// TIA Portal project "Project_Axe" (V15)

(* hardware
DEVICE "HMI_1"  KTP400 Basic mono PN
   slot 0: "HMI_1"  KTP400 Basic mono PN  6AV6 647-0AA11-3AX0  12.0.0.0
   slot 1: "HMI_RT_1"  KTP400 Basic mono PN  6AV6 647-0AA11-3AX0  12.0.0.0
   slot 5: "HMI_1.IE_CP_1"  PROFINET Interface  12.0.0.0
      slot 1: "PROFINET Interface_1"  PROFINET Interface
         slot 1: "Port_1"  Port
DEVICE "S7-1200 station_1"  S7-1200 Station
   slot 0: "Rack_0"  S7-1200 Rack  Rack  V1.0
   slot 1: "PLC"  CPU 1212C AC/DC/Rly  6ES7 212-1BE31-0XB0  V3.0
*)

// ===== PLC "PLC"  CPU 1212C AC/DC/Rly =====

VAR_GLOBAL   // PLC tag table "Default tag table"
   "All_SelectionsCorrect" AT %I100.0 : Bool;
   "Stop" AT %I100.1 : Bool;
   "AxeBack" AT %Q100.0 : Bool;
   "TreeFall" AT %Q100.1 : Bool;
   "Reset" AT %Q100.2 : Bool;
   "SelectionsCorrectLight" AT %Q100.3 : Bool;
END_VAR

DATA_BLOCK "G"   // DB1
{ S7_Optimized_Access := 'TRUE' }
VERSION : 0.1
   VAR
      T1_DwellTime : IEC_TIMER;
      T2_AxeBack : IEC_TIMER;
      T3_AxeBounce : IEC_TIMER;
      T4_AxeSwing : IEC_TIMER;
      T5_TreeFall : IEC_TIMER;
      T6_WatchDog : IEC_TIMER;
      ResetTimeDelay : IEC_TIMER;
   END_VAR
   VAR RETAIN
      HMI_T1_Time : Real := 10.0;
      HMI_T2_Time : Real := 10.0;
      HMI_T3_Time : Real := 10.0;
      HMI_T4_Time : Real := 10.0;
      HMI_T5_Time : Real := 10.0;
      HMI_T6_Time : Real := 10.0;
   END_VAR
   VAR
      T1_Time : DInt;
      T2_Time : DInt;
      T3_Time : DInt;
      T4_Time : DInt;
      T5_Time : DInt;
      T6_Time : DInt;
   END_VAR
BEGIN
END_DATA_BLOCK

FUNCTION "Timers" : Void   // FC1, LAD
{ S7_Optimized_Access := 'TRUE' }
VERSION : 0.1
   VAR_TEMP
      temp_real1 : Real;
      temp_real2 : Real;
      temp_real4 : Real;
      temp_real3 : Real;
      temp_real5 : Real;
      temp_real6 : Real;
      temp_real_sum : Real;
   END_VAR
   VAR_TEMP   // added for the SCL form of the ladder/FBD networks
      _w1 : Bool;
   END_VAR
BEGIN

REGION Network 1: Dwell Time Before Starting Cycle
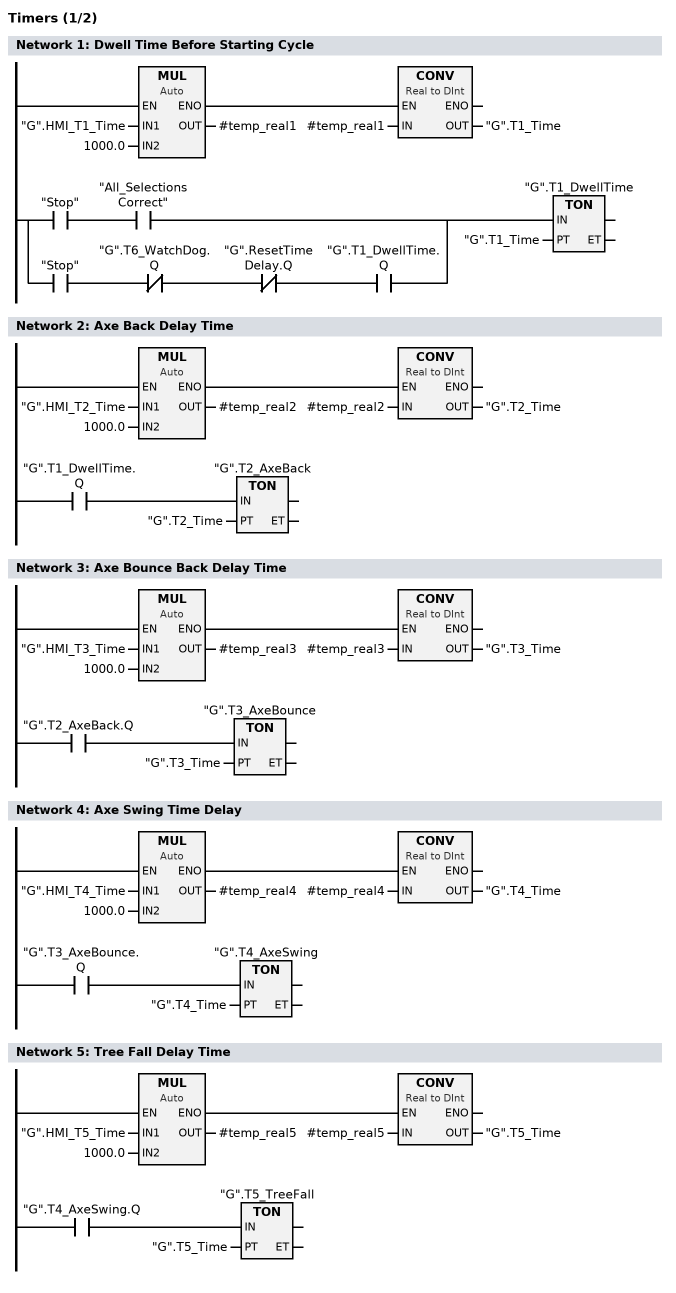
   // ENO of a box is taken as its EN; it also drops when the box reports an error
   #temp_real1 := "G".HMI_T1_Time * 1000.0;
   "G".T1_Time := REAL_TO_DINT(#temp_real1);
   "G".T1_DwellTime.TON(IN := ("Stop" AND "All_SelectionsCorrect") OR ("Stop" AND NOT "G".T6_WatchDog.Q AND NOT "G".ResetTimeDelay.Q AND "G".T1_DwellTime.Q),
                        PT := "G".T1_Time);
END_REGION

REGION Network 2: Axe Back Delay Time
   // ENO of a box is taken as its EN; it also drops when the box reports an error
   #temp_real2 := "G".HMI_T2_Time * 1000.0;
   "G".T2_Time := REAL_TO_DINT(#temp_real2);
   "G".T2_AxeBack.TON(IN := "G".T1_DwellTime.Q, PT := "G".T2_Time);
END_REGION

REGION Network 3: Axe Bounce Back Delay Time
   // ENO of a box is taken as its EN; it also drops when the box reports an error
   #temp_real3 := "G".HMI_T3_Time * 1000.0;
   "G".T3_Time := REAL_TO_DINT(#temp_real3);
   "G".T3_AxeBounce.TON(IN := "G".T2_AxeBack.Q, PT := "G".T3_Time);
END_REGION

REGION Network 4: Axe Swing Time Delay
   // ENO of a box is taken as its EN; it also drops when the box reports an error
   #temp_real4 := "G".HMI_T4_Time * 1000.0;
   "G".T4_Time := REAL_TO_DINT(#temp_real4);
   "G".T4_AxeSwing.TON(IN := "G".T3_AxeBounce.Q, PT := "G".T4_Time);
END_REGION

REGION Network 5: Tree Fall Delay Time
   // ENO of a box is taken as its EN; it also drops when the box reports an error
   #temp_real5 := "G".HMI_T5_Time * 1000.0;
   "G".T5_Time := REAL_TO_DINT(#temp_real5);
   "G".T5_TreeFall.TON(IN := "G".T4_AxeSwing.Q, PT := "G".T5_Time);
END_REGION

REGION Network 6: Watch Dog Delay Time. Summation of all times and the relay reset delay of 5 seconds
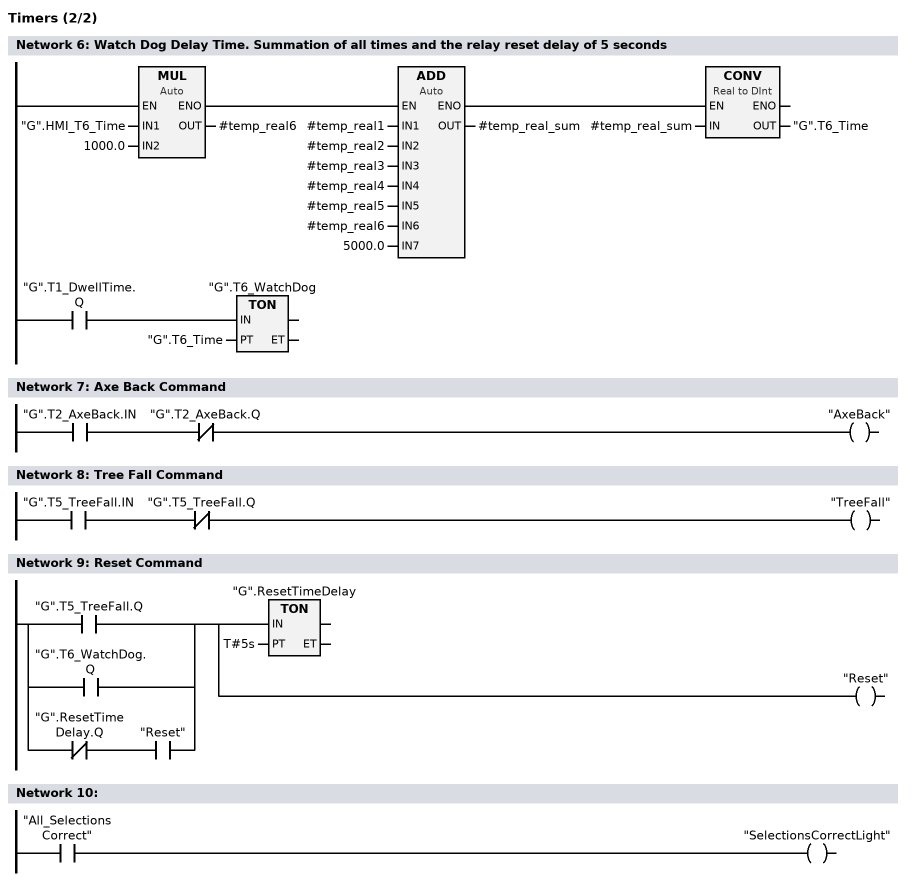
   // ENO of a box is taken as its EN; it also drops when the box reports an error
   #temp_real6 := "G".HMI_T6_Time * 1000.0;
   #temp_real_sum := #temp_real1 + #temp_real2 + #temp_real3 + #temp_real4 + #temp_real5 + #temp_real6 + 5000.0;
   "G".T6_Time := REAL_TO_DINT(#temp_real_sum);
   "G".T6_WatchDog.TON(IN := "G".T1_DwellTime.Q, PT := "G".T6_Time);
END_REGION

REGION Network 7: Axe Back Command
   RUNG wire#powerrail
      Contact( "G".T2_AxeBack.IN )
      I_Contact( "G".T2_AxeBack.Q )
      Coil( "AxeBack" )
   END_RUNG
   // the same network as SCL:
   "AxeBack" := "G".T2_AxeBack.IN AND NOT "G".T2_AxeBack.Q;
END_REGION

REGION Network 8: Tree Fall Command
   RUNG wire#powerrail
      Contact( "G".T5_TreeFall.IN )
      I_Contact( "G".T5_TreeFall.Q )
      Coil( "TreeFall" )
   END_RUNG
   // the same network as SCL:
   "TreeFall" := "G".T5_TreeFall.IN AND NOT "G".T5_TreeFall.Q;
END_REGION

REGION Network 9: Reset Command
   #_w1 := "G".T5_TreeFall.Q OR "G".T6_WatchDog.Q OR (NOT "G".ResetTimeDelay.Q AND "Reset");
   "G".ResetTimeDelay.TON(IN := #_w1, PT := T#5s);
   "Reset" := #_w1;
END_REGION

REGION Network 10
   RUNG wire#powerrail
      Contact( "All_SelectionsCorrect" )
      Coil( "SelectionsCorrectLight" )
   END_RUNG
   // the same network as SCL:
   "SelectionsCorrectLight" := "All_SelectionsCorrect";
END_REGION
END_FUNCTION

ORGANIZATION_BLOCK "Main"   // OB1, LAD, ProgramCycle
TITLE = "Main Program Sweep (Cycle)"
{ S7_Optimized_Access := 'TRUE' }
VERSION : 0.1
BEGIN

REGION Network 1
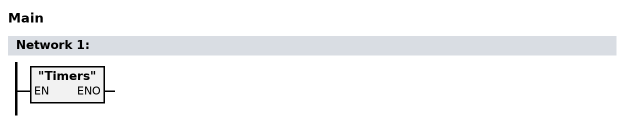
   RUNG wire#powerrail
      "Timers"()
   END_RUNG
   // the same network as SCL:
   "Timers"();
END_REGION
END_ORGANIZATION_BLOCK

(* ===== HMI "HMI_RT_1" =====
system functions are stored by id; their names below are inferred from use
connection "HMI_Connection_1": ETHERNET, SMART_S7_1200_OMS

HMI tags "Default tag table"
   "Tag_ScreenNumber" : UInt, internal
   "G_HMI_T1_Time" : Real = PLC G.HMI_T1_Time, 1 s
   "G_HMI_T2_Time" : Real = PLC G.HMI_T2_Time, 1 s
   "G_HMI_T3_Time" : Real = PLC G.HMI_T3_Time, 1 s
   "G_HMI_T4_Time" : Real = PLC G.HMI_T4_Time, 1 s
   "G_HMI_T5_Time" : Real = PLC G.HMI_T5_Time, 1 s
   "G_HMI_T6_Time" : Real = PLC G.HMI_T6_Time, 1 s
   "All_SelectionsCorrect" : Bool = PLC All_SelectionsCorrect AT %I100.0, 1 s
   "Stop" : Bool = PLC Stop AT %I100.1, 1 s
   "AxeBack" : Bool = PLC AxeBack AT %Q100.0, 1 s
   "TreeFall" : Bool = PLC TreeFall AT %Q100.1, 1 s
   "Reset" : Bool = PLC Reset AT %Q100.2, 1 s
   "G_T1_DwellTime.IN" : Bool = PLC G.T1_DwellTime.IN, 1 s
   "G_T1_DwellTime.Q" : Bool = PLC G.T1_DwellTime.Q, 1 s
   "G_T2_AxeBack.IN" : Bool = PLC G.T2_AxeBack.IN, 1 s
   "G_T2_AxeBack.Q" : Bool = PLC G.T2_AxeBack.Q, 1 s
   "G_T3_AxeBounce.IN" : Bool = PLC G.T3_AxeBounce.IN, 1 s
   "G_T3_AxeBounce.Q" : Bool = PLC G.T3_AxeBounce.Q, 1 s
   "G_T4_AxeSwing.IN" : Bool = PLC G.T4_AxeSwing.IN, 1 s
   "G_T4_AxeSwing.Q" : Bool = PLC G.T4_AxeSwing.Q, 1 s
   "G_T5_TreeFall.IN" : Bool = PLC G.T5_TreeFall.IN, 1 s
   "G_T5_TreeFall.Q" : Bool = PLC G.T5_TreeFall.Q, 1 s
   "G_T6_WatchDog.IN" : Bool = PLC G.T6_WatchDog.IN, 1 s
   "G_T6_WatchDog.Q" : Bool = PLC G.T6_WatchDog.Q, 1 s
   "SelectionsCorrectLight" : Bool = PLC SelectionsCorrectLight AT %Q100.3, 1 s

Template "Template_1" 320x240
   Softkey "Softkey_F1" at 0,0 size 0x0
      on KeyDown: ActivateScreen("Splash", 0)
   Softkey "Softkey_F2" at 0,0 size 0x0
      on KeyDown: ActivateScreen("Timers", 0)
   Softkey "Softkey_F3" at 0,0 size 0x0
      on KeyDown: ActivateScreen("Sequence", 0)
   Softkey "Softkey_F4" at 0,0 size 0x0
      on KeyDown: ActivateScreen("Screen4", 0)

screen "Splash" 320x240, template "Template_1"
   on GenerateScreen: SetTag("Tag_ScreenNumber", 1)
   TextField "Text Field_3" at 100,90 size 132x40; Text 'Paul's AXE'

screen "Sequence" 320x240
   TextField "Text Field_3" at 30,100 size 100x30; Text 'T1 Timing'
      Visibility <- "G_T1_DwellTime.IN"
   TextField "Text Field_1" at 30,10 size 100x30; Text 'Input 0'
      Visibility <- "All_SelectionsCorrect"
   TextField "Text Field_2" at 30,30 size 100x30; Text 'Input 1'
      Visibility <- "Stop"
   TextField "Text Field_5" at 30,120 size 100x30; Text 'T1 Done'
      Visibility <- "G_T1_DwellTime.Q"
   TextField "Text Field_6" at 30,140 size 100x30; Text 'T2 Timing'
      Visibility <- "G_T2_AxeBack.IN"
   TextField "Text Field_7" at 30,160 size 100x30; Text 'T2 Done'
      Visibility <- "G_T2_AxeBack.Q"
   TextField "Text Field_8" at 30,180 size 100x30; Text 'T3 Timing'
      Visibility <- "G_T3_AxeBounce.IN"
   TextField "Text Field_9" at 30,200 size 100x30; Text 'T3 Done'
      Visibility <- "G_T3_AxeBounce.Q"
   TextField "Text Field_10" at 180,100 size 100x30; Text 'T4 Timing'
      Visibility <- "G_T4_AxeSwing.IN"
   TextField "Text Field_11" at 180,120 size 100x30; Text 'T4 Done'
      Visibility <- "G_T4_AxeSwing.Q"
   TextField "Text Field_12" at 180,140 size 100x30; Text 'T5 Timing'
      Visibility <- "G_T5_TreeFall.IN"
   TextField "Text Field_13" at 180,160 size 100x30; Text 'T5 Done'
      Visibility <- "G_T5_TreeFall.Q"
   TextField "Text Field_14" at 180,180 size 100x30; Text 'T6 Timing'
      Visibility <- "G_T6_WatchDog.IN"
   TextField "Text Field_15" at 180,200 size 100x30; Text 'T6 Done'
      Visibility <- "G_T6_WatchDog.Q"
   TextField "Text Field_4" at 180,10 size 100x30; Text 'Output 0'
      Visibility <- "AxeBack"
   TextField "Text Field_16" at 180,30 size 100x30; Text 'Output 1'
      Visibility <- "TreeFall"
   TextField "Text Field_17" at 180,50 size 100x30; Text 'Output 2'
      Visibility <- "Reset"
   TextField "Text Field_18" at 180,70 size 100x30; Text 'Output 3'
      Visibility <- "SelectionsCorrectLight"
   Softkey "Softkey_F1" at 0,0 size 0x0
      on KeyDown: ActivateScreen("Splash", 0)
   Softkey "Softkey_F2" at 0,0 size 0x0
      on KeyDown: ActivateScreen("Timers", 0)
   Softkey "Softkey_F4" at 0,0 size 0x0
      on KeyDown: ActivateScreen("Screen4", 0)

screen "Screen4" 320x240
   Softkey "Softkey_F1" at 0,0 size 0x0
      on KeyDown: ActivateScreen("Splash", 0)
   Softkey "Softkey_F2" at 0,0 size 0x0
      on KeyDown: ActivateScreen("Timers", 0)
   Softkey "Softkey_F3" at 0,0 size 0x0
      on KeyDown: ActivateScreen("Sequence", 0)

screen "Timers" 320x240
   IOField "IO Field_2" at 210,0 size 68x30; FormatPattern 99.9
      ProcessValue <- "G_HMI_T1_Time"
   TextField "Text Field_3" at 40,0 size 172x30; Text 'T1 Dwell Time'
   IOField "IO Field_1" at 210,40 size 68x30; FormatPattern 99.9
      ProcessValue <- "G_HMI_T2_Time"
   TextField "Text Field_1" at 40,40 size 172x30; Text 'T2 Axe Back'
   IOField "IO Field_3" at 210,80 size 68x30; FormatPattern 99.9
      ProcessValue <- "G_HMI_T3_Time"
   TextField "Text Field_2" at 40,80 size 172x30; Text 'T3 Axe Bounce'
   IOField "IO Field_4" at 210,120 size 68x30; FormatPattern 99.9
      ProcessValue <- "G_HMI_T4_Time"
   TextField "Text Field_4" at 40,120 size 172x30; Text 'T4 Axe Swing'
   IOField "IO Field_5" at 210,160 size 68x30; FormatPattern 99.9
      ProcessValue <- "G_HMI_T5_Time"
   TextField "Text Field_5" at 40,160 size 172x30; Text 'T5 Tree Fall'
   IOField "IO Field_6" at 210,200 size 68x30; FormatPattern 99.9
      ProcessValue <- "G_HMI_T6_Time"
   TextField "Text Field_6" at 40,200 size 172x30; Text 'T6 Watch Dog'
   Softkey "Softkey_F1" at 0,0 size 0x0
      on KeyDown: ActivateScreen("Splash", 0)
   Softkey "Softkey_F3" at 0,0 size 0x0
      on KeyDown: ActivateScreen("Sequence", 0)
   Softkey "Softkey_F4" at 0,0 size 0x0
      on KeyDown: ActivateScreen("Screen4", 0)
*)